{attribute addProperty BoxType "EK1100-0000-0018"}
{attribute addProperty Id "Beckhoff_ELM36xxEK1122Beckhoff_ELM36xxEK1122_DABD45E4162A_0001_ELM3602_0000_0017ELM3602_1C598C2535244A_0002_ELM3602_0000_0018ELM3602_1C598C2535244A_0003_ELM3602_0002_0016ELM3602_1C598C2535244A_0004_ELM3602_0002_0017ELM3602_1C598C2535244A_0005_ELM3602_0002_0018ELM3602_1C598C2535244A_0006_ELM3604_0000_0017ELM3604_EF18820948060A_0007_ELM3604_0000_0018ELM3604_EF18820948060A_0008_ELM3604_0002_0016ELM3604_EF18820948060A_0009_ELM3604_0002_0017ELM3604_EF18820948060A_0010_ELM3604_0002_0018ELM3604_EF18820948060"}
{attribute addProperty CRC "827123901"}
{attribute addProperty SizeInBites "4176"}
{attribute addProperty SizeInBytes "522"}
TYPE Beckhoff_ELM36xx_314CE8BD EXTENDS EK1100_179A0949 :
STRUCT
	{attribute addProperty Name "Beckhoff_ELM36xxEK1122"}
	Beckhoff_ELM36xxEK1122 : Beckhoff_ELM36xxEK1122_DABD45E4;
	{attribute addProperty Name "A_0001_ELM3602_0000_0017"}
	A_0001_ELM3602_0000_0017 : ELM3602_1C598C25;
	{attribute addProperty Name "A_0002_ELM3602_0000_0018"}
	A_0002_ELM3602_0000_0018 : ELM3602_1C598C25;
	{attribute addProperty Name "A_0003_ELM3602_0002_0016"}
	A_0003_ELM3602_0002_0016 : ELM3602_1C598C25;
	{attribute addProperty Name "A_0004_ELM3602_0002_0017"}
	A_0004_ELM3602_0002_0017 : ELM3602_1C598C25;
	{attribute addProperty Name "A_0005_ELM3602_0002_0018"}
	A_0005_ELM3602_0002_0018 : ELM3602_1C598C25;
	{attribute addProperty Name "A_0006_ELM3604_0000_0017"}
	A_0006_ELM3604_0000_0017 : ELM3604_EF188209;
	{attribute addProperty Name "A_0007_ELM3604_0000_0018"}
	A_0007_ELM3604_0000_0018 : ELM3604_EF188209;
	{attribute addProperty Name "A_0008_ELM3604_0002_0016"}
	A_0008_ELM3604_0002_0016 : ELM3604_EF188209;
	{attribute addProperty Name "A_0009_ELM3604_0002_0017"}
	A_0009_ELM3604_0002_0017 : ELM3604_EF188209;
	{attribute addProperty Name "A_0010_ELM3604_0002_0018"}
	A_0010_ELM3604_0002_0018 : ELM3604_EF188209;
END_STRUCT
END_TYPE

(* stored: Version 1.2.0.0, ProductVersion 3.1.4024.9
   DUT Beckhoff_ELM36xx_314CE8BD: Id {0cbc499b-3d9e-4602-a69b-2381790ce0c6} *)
